TYPE eDirection : 
(
    MC_Positive_Direction := 1,
    MC_Shortest_Way := 2,
    MC_Negative_Direction := 3,
    MC_Current_Direction := 4,
    MC_Undefined_Direction := 128
) INT;
END_TYPE

(* stored: Version 1.1.0.1, ProductVersion 3.1.4024.6
   DUT eDirection: Id {aa1af5d3-a2aa-06ff-337e-445ad26c3677} *)
